// TIA Portal project "default_project" (V15.1)

(* hardware
DEVICE "S7-1200 station_1"  S7-1200 Station
   slot 0: "Rack_0"  S7-1200 Rack  Rack  V1.0
   slot 1: "PLC_1"  CPU 1214C DC/DC/DC  6ES7 214-1AG40-0XB0  V4.2
*)

// ===== PLC "PLC_1"  CPU 1214C DC/DC/DC =====

VAR_GLOBAL   // PLC tag table "Default tag table"
   "bt_open_gate" AT %I9.3 : Bool;
   "gate_opening" AT %Q1.6 : Bool;
   "bt_close_gate" AT %I9.4 : Bool;
   "gate_closing" AT %Q1.7 : Bool;
   "sensor_fdc_avanco" AT %I6.3 : Bool;
   "sensor_fdc_recuo" AT %I6.4 : Bool;
   "botao_parar" AT %I9.6 : Bool;
END_VAR

ORGANIZATION_BLOCK "Main"   // OB1, LAD, ProgramCycle
TITLE = "Main Program Sweep (Cycle)"
{ S7_Optimized_Access := 'TRUE' }
VERSION : 0.1
   VAR_INPUT
      Initial_Call : Bool;   // Initial call of this OB
      Remanence : Bool;   // =True, if remanent data are available
   END_VAR
BEGIN

REGION Network 1: Opening
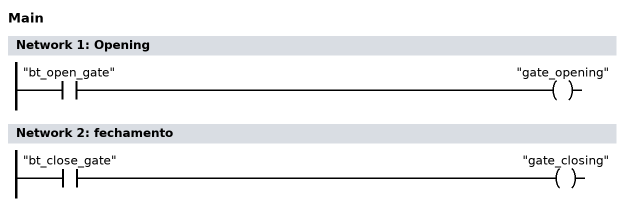
   RUNG wire#powerrail
      Contact( "bt_open_gate" )
      Coil( "gate_opening" )
   END_RUNG
   // the same network as SCL:
   "gate_opening" := "bt_open_gate";
END_REGION

REGION Network 2: fechamento
   RUNG wire#powerrail
      Contact( "bt_close_gate" )
      Coil( "gate_closing" )
   END_RUNG
   // the same network as SCL:
   "gate_closing" := "bt_close_gate";
END_REGION
END_ORGANIZATION_BLOCK